(* IEC 61131-3 sources: AXOpen/src/showcase/app/src/components.balluff.identification/Documentation, 5 files *)

(* ---- Axo_BIS_M_4XX_045.st ---- *)
USING AXOpen.Core;

NAMESPACE AXOpen.Components.Balluff.Identification
    {S7.extern=ReadWrite}
    CLASS Axo_BIS_M_4XX_045_Example EXTENDS AXOpen.Core.AxoObject
        //<ComponentDeclaration>
        VAR PUBLIC
            ExampleReader : AXOpen.Components.Balluff.Identification.Axo_BIS_M_4XX_045;
        END_VAR
        //</ComponentDeclaration>

        //<InitializationArgumentsDeclaration>
        VAR PUBLIC
            {#ix-set:AttributeName = "<#Activate manual control#>"}
            ActivateManualControl : BOOL;
        END_VAR
        //</InitializationArgumentsDeclaration>

        METHOD PUBLIC OVERRIDE Run
            VAR_INPUT
                inParent : IAxoObject;
            END_VAR

            SUPER.Run(inParent);

            IF ActivateManualControl THEN
                ExampleReader.ActivateManualControl();
            END_IF;

            //<Initialization>
            ExampleReader.Run(  inParent := THIS,
                                hwID     := AXOpen.Showcase.HwIdentifiers#BNIPNT507005Z040_HwID);
            //</Initialization>

            THIS.UseInSequencer();
        END_METHOD

        //<Usage>
        VAR PUBLIC
            Sequencer : AxoSequencer;
            Steps     : ARRAY[0..7] OF AXOpen.Core.AxoStep;
        END_VAR

        METHOD PRIVATE UseInSequencer

            Sequencer.Run(THIS);
            Sequencer.Open();
            Sequencer.SequenceMode := eAxoSequenceMode#RunOnce;

            IF(Steps[0].Execute(Sequencer, 'Configure and restore reader')) THEN
                ExampleReader.Config.InfoTime      := LTIME#2S;
                ExampleReader.Config.ErrorTime     := LTIME#5S;
                ExampleReader.Config.TaskTimeout   := LTIME#50S;
                ExampleReader.Config.StartAddress  := WORD#0;
                ExampleReader.Config.RfidCodeSize  := WORD#50;
                ExampleReader.Restore();
                Sequencer.MoveNext();
            END_IF;

            IF(Steps[1].Execute(Sequencer, 'Reset reader')) THEN
                IF(ExampleReader.ResetReader().IsDone()) THEN
                    Sequencer.MoveNext();
                END_IF;
            END_IF;

            IF(Steps[2].Execute(Sequencer, 'Read tag data')) THEN
                IF(ExampleReader.Read().IsDone()) THEN
                    Sequencer.MoveNext();
                END_IF;
            END_IF;

            IF(Steps[3].Execute(Sequencer, 'Write tag data')) THEN
                IF(ExampleReader.Write().IsDone()) THEN
                    Sequencer.MoveNext();
                END_IF;
            END_IF;

            IF(Steps[4].Execute(Sequencer, 'Write single char to memory')) THEN
                IF(ExampleReader.WriteCharToMemory(character     := BYTE#16#41,  // 'A'
                                                   Address       := WORD#0,
                                                   NumberOfBytes := WORD#1
                                                   ).IsDone()) THEN
                    Sequencer.MoveNext();
                END_IF;
            END_IF;

            IF(Steps[5].Execute(Sequencer, 'Reset communication')) THEN
                IF(ExampleReader.ResetCommunication().IsDone()) THEN
                    Sequencer.MoveNext();
                END_IF;
            END_IF;

            IF(Steps[6].Execute(Sequencer, 'Error recovery')) THEN
                ExampleReader.Restore();
                Sequencer.MoveNext();
            END_IF;

            IF(Steps[7].Execute(Sequencer, 'Complete')) THEN
                Sequencer.CompleteSequence();
            END_IF;
        END_METHOD
        //</Usage>
    END_CLASS
END_NAMESPACE

(* ---- Axo_BIS_M_4XX_045_ManualControl.st ---- *)
USING AXOpen.Core;

NAMESPACE AXOpen.Components.Balluff.Identification
    {S7.extern=ReadWrite}
    CLASS Axo_BIS_M_4XX_045_ManualControl_Example EXTENDS AXOpen.Core.AxoObject
        //<ComponentDeclaration>
        VAR PUBLIC
            ManualReader : AXOpen.Components.Balluff.Identification.Axo_BIS_M_4XX_045;
        END_VAR
        //</ComponentDeclaration>

        //<InitializationArgumentsDeclaration>
        VAR PUBLIC
            {#ix-set:AttributeName = "<#Activate manual control#>"}
            ActivateManualControl : BOOL := TRUE;
        END_VAR
        //</InitializationArgumentsDeclaration>

        METHOD PUBLIC OVERRIDE Run
            VAR_INPUT
                inParent : IAxoObject;
            END_VAR

            SUPER.Run(inParent);

            // In manual-control mode the operator drives individual tasks from
            // the HMI. Configuration is still applied from ST on startup.
            IF ActivateManualControl THEN
                ManualReader.ActivateManualControl();
            END_IF;

            //<Initialization>
            ManualReader.Config.InfoTime      := LTIME#2S;
            ManualReader.Config.ErrorTime     := LTIME#5S;
            ManualReader.Config.TaskTimeout   := LTIME#50S;
            ManualReader.Config.StartAddress  := WORD#0;
            ManualReader.Config.RfidCodeSize  := WORD#50;

            ManualReader.Run(  inParent := THIS,
                               hwID     := AXOpen.Showcase.HwIdentifiers#BNIPNT507005Z040_HwID);
            //</Initialization>

            IF NOT ActivateManualControl THEN
                ManualReader.Restore();
            END_IF;
        END_METHOD

        //<Usage>
        // This scenario has no sequencer -- the reader is operated entirely
        // from the RenderableContentControl (Command-Control presentation):
        //   * Restore             -- applies Config and clears errors
        //   * Read                -- triggers ReadTask on the connected tag
        //   * Write               -- triggers WriteTask with the configured payload
        //   * ResetReader         -- restarts the reader firmware
        //   * ResetCommunication  -- restarts the PROFINET communication channel
        //   * WriteCharToMemory   -- writes a single byte at a configurable address
        //</Usage>
    END_CLASS
END_NAMESPACE

(* ---- Axo_BIS_M_4XX_045_Showcase.st ---- *)
USING AXOpen.Core;

NAMESPACE AXOpen.Components.Balluff.Identification
    {S7.extern=ReadWrite}
    CLASS Axo_BIS_M_4XX_045_Showcase EXTENDS AXOpen.Core.AxoObject
        //<ComponentDeclaration>
        VAR PUBLIC
            ExampleReader : AXOpen.Components.Balluff.Identification.Axo_BIS_M_4XX_045;
        END_VAR
        //</ComponentDeclaration>

        //<InitializationArgumentsDeclaration>
        VAR PUBLIC
            {#ix-set:AttributeName = "<#Activate manual control#>"}
            ActivateManualControl : BOOL;
        END_VAR
        //</InitializationArgumentsDeclaration>

        METHOD PUBLIC OVERRIDE Run
            VAR_INPUT
                inParent : IAxoObject;
            END_VAR

            SUPER.Run(inParent);

            IF ActivateManualControl THEN
                ExampleReader.ActivateManualControl();
            END_IF;

            //<Initialization>
            ExampleReader.Run(  inParent := THIS,
                                hwID            := AXOpen.Showcase.HwIdentifiers#BNIPNT507005Z040_HwID);
            //</Initialization>

        THIS.UseInSequencer();
        END_METHOD

        //<Usage>
        VAR PUBLIC
            Sequencer : AxoSequencer;
            Steps : ARRAY[0..3] OF AXOpen.Core.AxoStep;
        END_VAR

        METHOD PRIVATE UseInSequencer

            Sequencer.Run(THIS);
            Sequencer.Open();

            IF(Steps[0].Execute(Sequencer, 'Read')) THEN
                IF(ExampleReader.Read().IsDone()) THEN
                    Sequencer.MoveNext();
                END_IF;
            END_IF;

            IF(Steps[1].Execute(Sequencer, 'Write')) THEN
                IF(ExampleReader.Write().IsDone()) THEN
                    Sequencer.MoveNext();
                END_IF;
            END_IF;
        END_METHOD

        //</Usage>
    END_CLASS
END_NAMESPACE

(* ---- Axo_BIS_M_4XX_045_Showcase2.st ---- *)
USING AXOpen.Core;

NAMESPACE AXOpen.Components.Balluff.Identification
    {S7.extern=ReadWrite}
    CLASS Axo_BIS_M_4XX_045_Showcase2 EXTENDS AXOpen.Core.AxoObject
        //<ComponentDeclaration>
        VAR PUBLIC
            ExampleReader : AXOpen.Components.Balluff.Identification.Axo_BIS_M_4XX_045;
        END_VAR
        //</ComponentDeclaration>

        //<InitializationArgumentsDeclaration>
        VAR PUBLIC
            {#ix-set:AttributeName = "<#Activate manual control#>"}
            ActivateManualControl : BOOL;
        END_VAR
        //</InitializationArgumentsDeclaration>

        METHOD PUBLIC OVERRIDE Run
            VAR_INPUT
                inParent : IAxoObject;
            END_VAR

            SUPER.Run(inParent);

            IF ActivateManualControl THEN
                ExampleReader.ActivateManualControl();
            END_IF;

            //<Initialization>
            ExampleReader.Run(  inParent := THIS,
                                hwID            := AXOpen.Showcase.HwIdentifiers#BNIPNT507005Z040_HwID);
            //</Initialization>

        THIS.UseInSequencer();
        END_METHOD

        //<Usage>
        VAR PUBLIC
            Sequencer : AxoSequencer;
            Steps : ARRAY[0..6] OF AXOpen.Core.AxoStep;
        END_VAR

        METHOD PRIVATE UseInSequencer

            Sequencer.Run(THIS);
            Sequencer.Open();
            Sequencer.SequenceMode := eAxoSequenceMode#RunOnce;

            IF(Steps[0].Execute(Sequencer, 'Restore')) THEN
                ExampleReader.Config.InfoTime      := LTIME#2S;
                ExampleReader.Config.ErrorTime     := LTIME#5S;
                ExampleReader.Config.TaskTimeout   := LTIME#50S;
                ExampleReader.Config.StartAddress  := WORD#0;
                ExampleReader.Config.RfidCodeSize  := WORD#50;
                ExampleReader.Restore();
                Sequencer.MoveNext();
            END_IF;

            IF(Steps[1].Execute(Sequencer, 'Reset reader')) THEN
                IF(ExampleReader.ResetReader().IsDone()) THEN
                    Sequencer.MoveNext();
                END_IF;
            END_IF;

            IF(Steps[2].Execute(Sequencer, 'Read')) THEN
                IF(ExampleReader.Read().IsDone()) THEN
                    Sequencer.MoveNext();
                END_IF;
            END_IF;

            IF(Steps[3].Execute(Sequencer, 'Write')) THEN
                IF(ExampleReader.Write().IsDone()) THEN
                    Sequencer.MoveNext();
                END_IF;
            END_IF;

            IF(Steps[4].Execute(Sequencer, 'Write char to memory')) THEN
                IF(ExampleReader.WriteCharToMemory(character     := BYTE#16#41,
                                                   Address       := WORD#0,
                                                   NumberOfBytes := WORD#1
                                                   ).IsDone()) THEN
                    Sequencer.MoveNext();
                END_IF;
            END_IF;

            IF(Steps[5].Execute(Sequencer, 'Reset communication')) THEN
                IF(ExampleReader.ResetCommunication().IsDone()) THEN
                    Sequencer.MoveNext();
                END_IF;
            END_IF;

            IF(Steps[6].Execute(Sequencer, 'Restore')) THEN
                ExampleReader.Restore();
                Sequencer.CompleteSequence();
            END_IF;
        END_METHOD

        //</Usage>
    END_CLASS
END_NAMESPACE

(* ---- BalluffIdentification.st ---- *)
NAMESPACE AXOpen.Components.Balluff.Identification
    {S7.extern=ReadWrite}
    CLASS BalluffIdentification EXTENDS AXOpen.Core.AxoObject
        VAR PUBLIC
            _rootObject : AxoObject;
            axo_BIS_M_4XX_045               : Axo_BIS_M_4XX_045_Example;
            axo_BIS_M_4XX_045_ManualControl : Axo_BIS_M_4XX_045_ManualControl_Example;
        END_VAR

        METHOD PUBLIC Execute
            _rootObject.Run(THIS);
            axo_BIS_M_4XX_045.Run(_rootObject);
            axo_BIS_M_4XX_045_ManualControl.Run(_rootObject);
        END_METHOD
    END_CLASS
END_NAMESPACE
